{attribute 'enable_dynamic_creation'}
FUNCTION_BLOCK FB_TargetTray EXTENDS FB_SlotTarget
VAR_INPUT
END_VAR
VAR_OUTPUT
END_VAR
VAR
END_VAR

METHOD FB_init : BOOL
VAR_INPUT
	bInitRetains : BOOL; // if TRUE, the retain variables are initialized (warm start / cold start)
	bInCopyCode : BOOL;  // if TRUE, the instance afterwards gets moved into the copy code (online change)
END_VAR
eObjectType := E_ObjectType.OBJECTTYPE_TargetTray;
eObjectGroup := E_ObjectGroup.OBJECTGROUP_Target;
END_METHOD

METHOD M_AddChild : ERRORID
VAR_INPUT
	pObject : POINTER TO FB_Object;
	nSlotNr	: UINT;
	nIndex 	: INT;
END_VAR
//Kann alle Targets aufnehmen
IF pObject > 0 THEN
	IF pObject^.M_bIsGroup(E_ObjectGroup.OBJECTGROUP_Target) THEN
		M_AddChild := SUPER^.M_AddChild(pObject,nSlotNr,nIndex);
	ELSE
		M_AddChild := E_ErrorIdObjMgmt.ERRORID_InvalidParentObject;
	END_IF
ELSE
	M_AddChild := E_ErrorIdObjMgmt.ERRORID_InvalidParentObject;
END_IF
END_METHOD

END_FUNCTION_BLOCK

(* stored: Version 1.1.0.1, ProductVersion 3.1.4022.18
   POU FB_TargetTray: Id {81d2859d-8093-4d0a-bb90-4254f7a1c91e}, SpecialFunc None
   Method FB_init: Id {5750d14d-e2f0-4891-b120-843e36e24e44}
   Method M_AddChild: Id {d1158298-0747-4b99-a9c0-c0cee68f8c91} *)
